FUNCTION_BLOCK FB_Component_Valve IMPLEMENTS I_Component
VAR_INPUT
	bSignal			: BOOL;				// Input valve
// Interface vars
	sName			: STRING[20];
	bEnable     	: BOOL;
	//eMode       	: E_ComponentMode;
END_VAR

VAR_OUTPUT
	bOutput			: BOOL;
	// interface vars
	eState			: E_ComponentState;
	iErrorCode		: INT;
	sStatusText 	: STRING[50];
END_VAR

IF 	bEnable AND (eState = E_ComponentState.READY OR eState = E_ComponentState.BUSY) THEN
	bOutput 	:= bSignal;
ELSE
	bOutput 	:= FALSE;
	sStatusText := 'Disabled';
END_IF

{warning 'add method implementation '}
METHOD Halt : BOOL
END_METHOD

{warning 'add method implementation '}
METHOD Start : BOOL
END_METHOD

{warning 'add method implementation '}
METHOD Stop : BOOL
END_METHOD

END_FUNCTION_BLOCK

(* stored: Version 1.1.0.1, ProductVersion 3.1.4024.15
   POU FB_Component_Valve: Id {e241cca9-8ad1-4d32-953d-80e7ad832e70}, SpecialFunc None
   Method Halt: Id {d6d164e4-6ff2-4655-bb53-7508a90ca844}
   Method Start: Id {3b5e4edb-f27f-4280-94ac-c799f1f4bcbc}
   Method Stop: Id {8f25114a-9d10-4e85-92e5-9d523c21fcd3} *)
